VISUALIZATION HarvStats  // 2x2
END_VISUALIZATION

(* stored: Version 1.1.0.1, ProductVersion 3.1.4024.15
   Visu HarvStats: Id {694051b8-c595-41e4-83e1-6d8a8cb35228} *)
